FUNCTION_BLOCK FB_GC_Module EXTENDS FB_ModuleBase
VAR_INPUT	
	HwInput : ST_GC_Signal_In;
	HwOutput : ST_GC_Signal_Out;

	ServiceCtrl : REFERENCE TO ST_GC_ServiceCtrl;
	ServiceParam : REFERENCE TO ST_GC_ServiceParam;

	// Base unit used in GC chamber
	SpinAxis_BaseUnit : I_Axis_BaseUnit;
	LiftPinAxis_BaseUnit : I_Axis_BaseUnit;
END_VAR

VAR_OUTPUT
	ServiceStatus : ST_GC_ServiceStatus;
END_VAR

VAR
	// 有需要特殊操作的需求，所以建立一個 ST_GC_ServiceCtrl 變數，讓程式內部可以過一手處理
	_ServiceCtrlView : U_GC_ServiceCtrlView;
	_ServiceStatusView : U_GC_ServiceStatusView;

	_nIdx : UINT;
	_SpinAxisJogCWService : FB_GCSpinAxisJogCWServices;
	_SpinAxisMoveAbsService : FB_GCSpinAxisMoveAbsServices;
	_SpinAxisMoveVelCWService : FB_GCSpinAxisMoveVelCWServices;
	_LiftPinAxisMoveVelCWService : FB_GCLiftPinAxisMoveVelCWServices;
	_LiftPinAxisMoveVelCCWService : FB_GCLiftPinAxisMoveVelCCWServices;
	_LiftPinAxisMoveAbsService : FB_GCLiftPinAxisMoveAbsServices;
	_SingleProcessService : FB_GCSingleProcessService;
	_SingleProcessStatus : ST_GCSingleProcessStatus;

	_VariableSimulationTick : DINT;
	_SimChamberTemperature : REAL;
	_SimChamberPressure : REAL;
END_VAR

// An unbound Axis interface is a composition error. Keep the Module inert.
IF (SpinAxis_BaseUnit = 0) OR (LiftPinAxis_BaseUnit = 0) THEN
	RETURN;
END_IF

M_UpdateModule();

// Updata status
ServiceStatus := _ServiceStatusView.ByName;

METHOD PROTECTED H_OnAborted
VAR_INPUT
	bFirstScan	: BOOL;
END_VAR
// Default action hook intentionally empty. Override in derived FBs when needed.
END_METHOD

METHOD PROTECTED H_OnAborting : E_PackMLHookResult
VAR_INPUT
	bFirstScan	: BOOL;
END_VAR
H_OnAborting := E_PackMLHookResult.Busy;

// Wait cmd finished
FOR _nIdx := 1 TO GVL_GC_Config.cServiceCount DO
	IF _ServiceStatusView.ByIndex[_nIdx].PackMLOut.eStateCurrent <> E_PackMLState.Aborted THEN
		RETURN;
	END_IF
END_FOR

H_OnAborting := E_PackMLHookResult.Done;
END_METHOD

METHOD PROTECTED H_OnClearing : E_PackMLHookResult
VAR_INPUT
	bFirstScan	: BOOL;
END_VAR
H_OnClearing := E_PackMLHookResult.Busy;

// Wait cmd finished
FOR _nIdx := 1 TO GVL_GC_Config.cServiceCount DO
	IF _ServiceStatusView.ByIndex[_nIdx].PackMLOut.eStateCurrent <> E_PackMLState.Stopped THEN
		RETURN;
	END_IF
END_FOR

H_OnClearing := E_PackMLHookResult.Done;
END_METHOD

METHOD PROTECTED H_OnComplete
VAR_INPUT
	bFirstScan	: BOOL;
END_VAR
// Default action hook intentionally empty. Override in derived FBs when needed.
END_METHOD

METHOD PROTECTED H_OnCompleting : E_PackMLHookResult
VAR_INPUT
	bFirstScan	: BOOL;
END_VAR
// Default transient hooks complete immediately; override when work is required.
H_OnCompleting := E_PackMLHookResult.Done;
END_METHOD

METHOD PROTECTED H_OnExecute : E_PackMLHookResult
VAR_INPUT
	bFirstScan	: BOOL;
END_VAR
// Execute is stable by default; derived FBs decide when the process is done.
H_OnExecute := E_PackMLHookResult.Busy;
END_METHOD

METHOD PROTECTED H_OnHeld
VAR_INPUT
	bFirstScan	: BOOL;
END_VAR
// Default action hook intentionally empty. Override in derived FBs when needed.
END_METHOD

METHOD PROTECTED H_OnHolding : E_PackMLHookResult
VAR_INPUT
	bFirstScan	: BOOL;
END_VAR
// Default transient hooks complete immediately; override when work is required.
H_OnHolding := E_PackMLHookResult.Done;
END_METHOD

METHOD PROTECTED H_OnIdle
VAR_INPUT
	bFirstScan	: BOOL;
END_VAR
// Default action hook intentionally empty. Override in derived FBs when needed.

// Transfer to execute automatically
RequestCommand(E_PackMLCommand.Start);
END_METHOD

METHOD PROTECTED H_OnResetting : E_PackMLHookResult
VAR_INPUT
	bFirstScan	: BOOL;
END_VAR
H_OnResetting := E_PackMLHookResult.Busy;

// Wait cmd finished
FOR _nIdx := 1 TO GVL_GC_Config.cServiceCount DO
	IF _ServiceStatusView.ByIndex[_nIdx].PackMLOut.eStateCurrent <> E_PackMLState.Idle THEN
		RETURN;
	END_IF
END_FOR

H_OnResetting := E_PackMLHookResult.Done;
END_METHOD

METHOD PROTECTED H_OnStarting : E_PackMLHookResult
VAR_INPUT
	bFirstScan	: BOOL;
END_VAR
// Default transient hooks complete immediately; override when work is required.
H_OnStarting := E_PackMLHookResult.Done;
END_METHOD

METHOD PROTECTED H_OnStopped
VAR_INPUT
	bFirstScan	: BOOL;
END_VAR
// Default action hook intentionally empty. Override in derived FBs when needed.
END_METHOD

METHOD PROTECTED H_OnStopping : E_PackMLHookResult
VAR_INPUT
	bFirstScan	: BOOL;
END_VAR
H_OnStopping := E_PackMLHookResult.Busy;

// Wait cmd finished
FOR _nIdx := 1 TO GVL_GC_Config.cServiceCount DO
	IF _ServiceStatusView.ByIndex[_nIdx].PackMLOut.eStateCurrent <> E_PackMLState.Stopped THEN
		RETURN;
	END_IF
END_FOR

H_OnStopping := E_PackMLHookResult.Done;
END_METHOD

METHOD PROTECTED H_OnSuspended
VAR_INPUT
	bFirstScan	: BOOL;
END_VAR
// Default action hook intentionally empty. Override in derived FBs when needed.
END_METHOD

METHOD PROTECTED H_OnSuspending : E_PackMLHookResult
VAR_INPUT
	bFirstScan	: BOOL;
END_VAR
// Default transient hooks complete immediately; override when work is required.
H_OnSuspending := E_PackMLHookResult.Done;
END_METHOD

METHOD PROTECTED H_OnUndefined : E_PackMLHookResult
VAR_INPUT
	bFirstScan	: BOOL;
END_VAR
// The base FB leaves Undefined immediately unless a derived FB delays startup.
H_OnUndefined := E_PackMLHookResult.Done;
END_METHOD

METHOD PROTECTED H_OnUnholding : E_PackMLHookResult
VAR_INPUT
	bFirstScan	: BOOL;
END_VAR
// Default transient hooks complete immediately; override when work is required.
H_OnUnholding := E_PackMLHookResult.Done;
END_METHOD

METHOD PROTECTED H_OnUnsuspending : E_PackMLHookResult
VAR_INPUT
	bFirstScan	: BOOL;
END_VAR
// Default transient hooks complete immediately; override when work is required.
H_OnUnsuspending := E_PackMLHookResult.Done;
END_METHOD

METHOD PROTECTED H_SelectServiceControlSource
VAR_INPUT
END_VAR
// Select control source
IF PackMLOut.eStateCurrent = E_PackMLState.Idle
	OR PackMLOut.eStateCurrent = E_PackMLState.Starting
	OR PackMLOut.eStateCurrent = E_PackMLState.Execute THEN
	// Controlled by external operator
	_ServiceCtrlView.ByName := ServiceCtrl;
ELSE
	// Control by module
	FOR _nIdx := 1 TO GVL_GC_Config.cServiceCount DO
		_ServiceCtrlView.ByIndex[_nIdx].PackMLIn := ModuleCtrl.PackMLIn;
		_ServiceCtrlView.ByIndex[_nIdx].RequestId := ModuleCtrl.RequestId;
	END_FOR
END_IF
END_METHOD

METHOD PROTECTED H_UpdateServiceAlarms
VAR_INPUT
END_VAR

VAR
	nServiceIndex : UINT;
	nErrorIndex : UINT;
END_VAR
// Submit the currently observable Service errors. The manager owns lifecycle state
// and marks identities not observed in this scan inactive during M_EndCycle.
FOR nServiceIndex := 1 TO GVL_GC_Config.cServiceCount DO
	FOR nErrorIndex := 1 TO Param_Config.MaxServiceError DO
		IF _ServiceStatusView.ByIndex[nServiceIndex].ErrorList[nErrorIndex].MainErrorId <> 0 THEN
			M_ObserveServiceAlarm(
				Alarm := _ServiceStatusView.ByIndex[nServiceIndex].ErrorList[nErrorIndex]);
		END_IF
	END_FOR
END_FOR
END_METHOD

METHOD PROTECTED H_UpdateBaseUnit
VAR_INPUT
END_VAR
SpinAxis_BaseUnit.M_CyclicUpdate();
LiftPinAxis_BaseUnit.M_CyclicUpdate();
END_METHOD

METHOD PROTECTED H_UpdateService
VAR_INPUT
END_VAR
_SpinAxisJogCWService(
	Ctrl:= _ServiceCtrlView.ByName.SpinAxisJogCW,
	Context:= _ServiceContext,
	Axis_BaseUnit:= SpinAxis_BaseUnit,
	// Owner IDs are assigned by the Module so each Service instance is unique.
	ServiceId:= E_GCServiceId.SpinAxisJogCW,
	Status=> _ServiceStatusView.ByName.SpinAxisJogCW);

_SpinAxisMoveAbsService(
	Ctrl:= _ServiceCtrlView.ByName.SpinAxisMoveAbs,
	Context:= _ServiceContext,
	Axis_BaseUnit:= SpinAxis_BaseUnit,
	ServiceId:= E_GCServiceId.SpinAxisMoveAbs,
	Status=> _ServiceStatusView.ByName.SpinAxisMoveAbs);

_SpinAxisMoveVelCWService(
	Ctrl:= _ServiceCtrlView.ByName.SpinAxisMoveVelCW,
	Context:= _ServiceContext,
	Axis_BaseUnit:= SpinAxis_BaseUnit,
	ServiceId:= E_GCServiceId.SpinAxisMoveVelCW,
	Status=> _ServiceStatusView.ByName.SpinAxisMoveVelCW);

_LiftPinAxisMoveVelCWService(
	Ctrl:= _ServiceCtrlView.ByName.LiftPinAxisMoveVelCW,
	Context:= _ServiceContext,
	Axis_BaseUnit:= LiftPinAxis_BaseUnit,
	ServiceId:= E_GCServiceId.LiftPinAxisMoveVelCW,
	Status=> _ServiceStatusView.ByName.LiftPinAxisMoveVelCW);

_LiftPinAxisMoveVelCCWService(
	Ctrl:= _ServiceCtrlView.ByName.LiftPinAxisMoveVelCCW,
	Context:= _ServiceContext,
	Axis_BaseUnit:= LiftPinAxis_BaseUnit,
	ServiceId:= E_GCServiceId.LiftPinAxisMoveVelCCW,
	Status=> _ServiceStatusView.ByName.LiftPinAxisMoveVelCCW);

_LiftPinAxisMoveAbsService(
	Ctrl:= _ServiceCtrlView.ByName.LiftPinAxisMoveAbs,
	Context:= _ServiceContext,
	Axis_BaseUnit:= LiftPinAxis_BaseUnit,
	ServiceId:= E_GCServiceId.LiftPinAxisMoveAbs,
	Status=> _ServiceStatusView.ByName.LiftPinAxisMoveAbs);

_SingleProcessService(
	Ctrl := _ServiceCtrlView.ByName.SingleProcess,
	Context := _ServiceContext,
	SpinAxis_BaseUnit := SpinAxis_BaseUnit,
	LiftPinAxis_BaseUnit := LiftPinAxis_BaseUnit,
	ServiceId := E_GCServiceId.SingleProcess,
	Status => _ServiceStatusView.ByName.SingleProcess,
	ProcessStatus => _SingleProcessStatus);
END_METHOD

METHOD PROTECTED H_UpdateServiceDataList
VAR_INPUT
END_VAR
VAR
	TimingView : U_GCSingleProcessStageTimingView;
	nIndex : UINT;
END_VAR
IF _SingleProcessStatus.LastCycle.Result <> E_GCSingleProcessResult.Completed THEN
	RETURN;
END_IF

TimingView.ByName := _SingleProcessStatus.LastCycle.StageTiming;
FOR nIndex := 1 TO 8 DO
	IF NOT TimingView.ByIndex[nIndex].Completed THEN
		RETURN;
	END_IF
END_FOR

// Replace the published snapshot only after a complete successful cycle.
MEMSET(ADR(ModuleDataList), 0, SIZEOF(ModuleDataList));
M_WriteStageServiceData(1, 'Prepare', TimingView.ByName.Prepare);
M_WriteStageServiceData(2, 'LiftReady', TimingView.ByName.LiftReady);
M_WriteStageServiceData(3, 'SpinAlign', TimingView.ByName.SpinAlign);
M_WriteStageServiceData(4, 'ConcurrentProcessEntry', TimingView.ByName.ConcurrentProcessEntry);
M_WriteStageServiceData(5, 'SpinRampUp', TimingView.ByName.SpinRampUp);
M_WriteStageServiceData(6, 'ProcessHold', TimingView.ByName.ProcessHold);
M_WriteStageServiceData(7, 'ConcurrentProcessExit', TimingView.ByName.ConcurrentProcessExit);
M_WriteStageServiceData(8, 'SpinStandby', TimingView.ByName.SpinStandby);
END_METHOD

METHOD PROTECTED H_UpdateServiceParam
VAR_INPUT
END_VAR
_SpinAxisMoveAbsService.Param := ServiceParam.SpinAxisMoveAbs;
_SpinAxisJogCWService.Param := ServiceParam.SpinAxisJogCW;
_SpinAxisMoveVelCWService.Param := ServiceParam.SpinAxisMoveVelCW;
_LiftPinAxisMoveVelCWService.Param := ServiceParam.LiftPinAxisMoveVelCW;
_LiftPinAxisMoveVelCCWService.Param := ServiceParam.LiftPinAxisMoveVelCCW;
_LiftPinAxisMoveAbsService.Param := ServiceParam.LiftPinAxisMoveAbs;
_SingleProcessService.Param := ServiceParam.SingleProcess;
END_METHOD

METHOD PRIVATE M_WriteStageServiceData
VAR_INPUT
	StageIndex : UINT;
	StageName : STRING(22);
	StageTiming : ST_GCSingleProcessStageTiming;
END_VAR
VAR
	nStartIndex : UINT;
	nEndIndex : UINT;
	nActualIndex : UINT;
END_VAR
nStartIndex := ((StageIndex - 1) * 3) + 1;
nEndIndex := nStartIndex + 1;
nActualIndex := nStartIndex + 2;

ModuleDataList[nStartIndex].Id := 700 + nStartIndex;
ModuleDataList[nStartIndex].Name := CONCAT(StageName, 'StartUtc');
ModuleDataList[nStartIndex].DataType := E_DescriptorType.DateTime;
ModuleDataList[nStartIndex].Unit := 'UTC';
ModuleDataList[nStartIndex].Value := StageTiming.StartUtc;

ModuleDataList[nEndIndex].Id := 700 + nEndIndex;
ModuleDataList[nEndIndex].Name := CONCAT(StageName, 'EndUtc');
ModuleDataList[nEndIndex].DataType := E_DescriptorType.DateTime;
ModuleDataList[nEndIndex].Unit := 'UTC';
ModuleDataList[nEndIndex].Value := StageTiming.EndUtc;

ModuleDataList[nActualIndex].Id := 700 + nActualIndex;
ModuleDataList[nActualIndex].Name := CONCAT(StageName, 'ActualMs');
ModuleDataList[nActualIndex].DataType := E_DescriptorType.Integer_32bit;
ModuleDataList[nActualIndex].Unit := 'ms';
ModuleDataList[nActualIndex].Value := DINT_TO_STRING(TIME_TO_DINT(StageTiming.ActualTime));
END_METHOD

END_FUNCTION_BLOCK

(* stored: Version 1.1.0.1, ProductVersion 3.1.4026.18
   POU FB_GC_Module: Id {d2b222b5-592d-46be-8a8e-fa50af509b93}, SpecialFunc None
   Folder ModuleUpdate: Id {a9f2fa3e-34f5-43fc-8823-0e0dbffba0ff}
   Folder StateAction: Id {92cfe23b-b998-4d76-8aa2-c8089e78aa61}
   Method H_OnAborted: Id {de8d6f56-427f-41df-b4d5-ddd289e1aed8}
   Method H_OnAborting: Id {29c05c7a-ae95-4991-b775-aae453451d8c}
   Method H_OnClearing: Id {b7069c3b-bd41-45c4-a177-00789e12f344}
   Method H_OnComplete: Id {9ab7169f-1450-41d3-b3d7-d608e72d68f0}
   Method H_OnCompleting: Id {6a295d34-cfdf-466f-b604-2e762f01df0b}
   Method H_OnExecute: Id {dc703a52-8c8a-4e2d-8deb-4adebb327ad6}
   Method H_OnHeld: Id {93f6b454-4398-4439-9237-4d01e13b7ccc}
   Method H_OnHolding: Id {d74d6d7d-e0fe-48fb-8a46-ad96f64e1fa5}
   Method H_OnIdle: Id {f9aa0f59-b1bb-45b6-82a2-3aac2bdc4e33}
   Method H_OnResetting: Id {f6ec54bd-ad3d-49c4-9547-ff474beb3546}
   Method H_OnStarting: Id {2befc923-f5b2-4ef5-aa0b-77c9a7b33520}
   Method H_OnStopped: Id {ce5006a2-3926-4be3-8c7a-d8efdde1ca29}
   Method H_OnStopping: Id {2d9e9bf2-b821-4b2d-9e15-b22384f79334}
   Method H_OnSuspended: Id {cff92aa7-0bee-4d5f-a95f-be0ba263ee0f}
   Method H_OnSuspending: Id {5fe72161-6df8-45fc-8c16-29aa2466b4be}
   Method H_OnUndefined: Id {c8ca4bd2-e69c-48f1-bbc8-42b473d6b552}
   Method H_OnUnholding: Id {64c7cdee-7a16-4239-96a0-6ebcc2d0e61c}
   Method H_OnUnsuspending: Id {c36273cc-b3d2-484e-a95e-475cdbf1ae08}
   Method H_SelectServiceControlSource: Id {4e055faf-6a98-4100-b6ed-93be619c0d1f}
   Method H_UpdateServiceAlarms: Id {05cb1d79-8999-497c-aa97-eff4f365f571}
   Method H_UpdateBaseUnit: Id {23db425b-9082-4959-8f76-43820da7ead4}
   Method H_UpdateService: Id {fa65f410-1990-4021-8134-1329f3f00eeb}
   Method H_UpdateServiceDataList: Id {0ea950db-71b5-4fd2-a9e8-c12c78c02390}
   Method H_UpdateServiceParam: Id {1a4b35b3-f132-467f-941f-899cd13c7e6b}
   Method M_WriteStageServiceData: Id {6f0188dd-ab9d-4b96-9248-74a942e61fd2} *)
